// TwinCAT 3 PLC project CM
// ProgramVersion: 3.1.4024.0
// libraries:
//   Tc2_ModbusRTU, * (Beckhoff Automation GmbH)
//   Tc2_Standard, * (Beckhoff Automation GmbH)
//   Tc2_System, * (Beckhoff Automation GmbH)
//   Tc2_Utilities, * (Beckhoff Automation GmbH)
//   Tc3_CM, * (Beckhoff Automation GmbH)
//   Tc3_CM_Base, * (Beckhoff Automation GmbH)
//   Tc3_Filter, * (Beckhoff Automation GmbH)
//   Tc3_Module, * (Beckhoff Automation GmbH)
//   Tc3_MultiArray, * (Beckhoff Automation GmbH)
// project tree:
//   DUTs/ E_AnalysisIDs.TcDUT, ST_HRErrHist.TcDUT
//   FBs/ FB_HRErrHist.TcPOU, FB_SystemTime.TcPOU
//   GVLs/ CM_Params.TcGVL, CM_Data.TcGVL, GVL_ADS.TcGVL, GVL_HMI.TcGVL, GVL_IO.TcGVL
//   / PlcTask.TcTTO, PlcTaskCM.TcTTO, TaskCalc.TcTTO
//   MAIN/ MAIN.TcPOU, MAIN_CM.TcPOU
//   PRGs/ PRG_Calculate.TcPOU, PRG_Database.TcPOU, PRG_Motor_Sensor.TcPOU
// real-time tasks:
//   TASK CMFast: cycle T#1ms, priority 4, ADS port 350
//   TASK CMSlow: cycle T#5ms, priority 12, ADS port 351
//   TASK PMFast: cycle T#1ms, priority 6, ADS port 352
//   TASK PMSlow: cycle T#10ms, priority 16, ADS port 353
//   TASK TaskCalc: cycle T#1ms, priority 8, ADS port 354
//   TASK EIPTask: cycle T#5ms, priority 1, ADS port 301
// I/O:
//   DEVICE Device 5 (EtherCAT) (disabled), AmsNetId 192.168.2.43.6.1
//     Term 1 (EK1100) [EK1100 EtherCAT Coupler (2A E-Bus)]
//       Term 2 (EL1094) [EL1094 4Ch. Dig. Input 24V, 10µs, negative]
//       Term 3 (EL3064) [EL3064 4Ch. Ana. Input 0-10V]
//       Term 4 (EL3632) [EL3632 2Ch. IEPE Sensor]
//       Term 5 (EL6021) [EL6021 Interface (RS422/485)]
//       Term 6 (EL3773) [EL3773 3 Ch. Power Monitoring, Oversample]
//       Term 7 (EL9011) [EL9011 End Terminal]
// variable links:
//   CM/CM Instance <-> Device 5 (EtherCAT)/Term 1 (EK1100)/Term 2 (EL1094)
//     PlcTaskCM Inputs/GVL_IO.bRev <-> Channel 1/Input
//   CM/CM Instance <-> Device 5 (EtherCAT)/Term 1 (EK1100)/Term 3 (EL3064)
//     PlcTaskCM Inputs/GVL_IO.iTemp <-> AI Standard Channel 1/Value
//   CM/CM Instance <-> Device 5 (EtherCAT)/Term 1 (EK1100)/Term 4 (EL3632)
//     PlcTask Inputs/GVL_IO.aEl3632[1][{1..10}] <-> Ch1 Sample {0..9}/Ch1 Value  (10 links)
//   PM/PM Instance <-> Device 5 (EtherCAT)/Term 1 (EK1100)/Term 6 (EL3773)
//     PlcTask Inputs/GVL.stEL3773_1_In/aIL1[10] <-> L1 Current Samples/I1 Samples[9]
//     PlcTask Inputs/GVL.stEL3773_1_In/aIL1[1] <-> L1 Current Samples/I1 Samples[0]
//     PlcTask Inputs/GVL.stEL3773_1_In/aIL1[2] <-> L1 Current Samples/I1 Samples[1]
//     PlcTask Inputs/GVL.stEL3773_1_In/aIL1[3] <-> L1 Current Samples/I1 Samples[2]
//     PlcTask Inputs/GVL.stEL3773_1_In/aIL1[4] <-> L1 Current Samples/I1 Samples[3]
//     PlcTask Inputs/GVL.stEL3773_1_In/aIL1[5] <-> L1 Current Samples/I1 Samples[4]
//     PlcTask Inputs/GVL.stEL3773_1_In/aIL1[6] <-> L1 Current Samples/I1 Samples[5]
//     PlcTask Inputs/GVL.stEL3773_1_In/aIL1[7] <-> L1 Current Samples/I1 Samples[6]
//     PlcTask Inputs/GVL.stEL3773_1_In/aIL1[8] <-> L1 Current Samples/I1 Samples[7]
//     PlcTask Inputs/GVL.stEL3773_1_In/aIL1[9] <-> L1 Current Samples/I1 Samples[8]
//     PlcTask Inputs/GVL.stEL3773_1_In/aIL2[10] <-> L2 Current Samples/I2 Samples[9]
//     PlcTask Inputs/GVL.stEL3773_1_In/aIL2[1] <-> L2 Current Samples/I2 Samples[0]
//     PlcTask Inputs/GVL.stEL3773_1_In/aIL2[2] <-> L2 Current Samples/I2 Samples[1]
//     PlcTask Inputs/GVL.stEL3773_1_In/aIL2[3] <-> L2 Current Samples/I2 Samples[2]
//     PlcTask Inputs/GVL.stEL3773_1_In/aIL2[4] <-> L2 Current Samples/I2 Samples[3]
//     PlcTask Inputs/GVL.stEL3773_1_In/aIL2[5] <-> L2 Current Samples/I2 Samples[4]
//     PlcTask Inputs/GVL.stEL3773_1_In/aIL2[6] <-> L2 Current Samples/I2 Samples[5]
//     PlcTask Inputs/GVL.stEL3773_1_In/aIL2[7] <-> L2 Current Samples/I2 Samples[6]
//     PlcTask Inputs/GVL.stEL3773_1_In/aIL2[8] <-> L2 Current Samples/I2 Samples[7]
//     PlcTask Inputs/GVL.stEL3773_1_In/aIL2[9] <-> L2 Current Samples/I2 Samples[8]
//     PlcTask Inputs/GVL.stEL3773_1_In/aIL3[10] <-> L3 Current Samples/I3 Samples[9]
//     PlcTask Inputs/GVL.stEL3773_1_In/aIL3[1] <-> L3 Current Samples/I3 Samples[0]
//     PlcTask Inputs/GVL.stEL3773_1_In/aIL3[2] <-> L3 Current Samples/I3 Samples[1]
//     PlcTask Inputs/GVL.stEL3773_1_In/aIL3[3] <-> L3 Current Samples/I3 Samples[2]
//     PlcTask Inputs/GVL.stEL3773_1_In/aIL3[4] <-> L3 Current Samples/I3 Samples[3]
//     PlcTask Inputs/GVL.stEL3773_1_In/aIL3[5] <-> L3 Current Samples/I3 Samples[4]
//     PlcTask Inputs/GVL.stEL3773_1_In/aIL3[6] <-> L3 Current Samples/I3 Samples[5]
//     PlcTask Inputs/GVL.stEL3773_1_In/aIL3[7] <-> L3 Current Samples/I3 Samples[6]
//     PlcTask Inputs/GVL.stEL3773_1_In/aIL3[8] <-> L3 Current Samples/I3 Samples[7]
//     PlcTask Inputs/GVL.stEL3773_1_In/aIL3[9] <-> L3 Current Samples/I3 Samples[8]
//     PlcTask Inputs/GVL.stEL3773_1_In/aUL1[10] <-> L1 Voltage Samples/U1 Samples[9]
//     PlcTask Inputs/GVL.stEL3773_1_In/aUL1[1] <-> L1 Voltage Samples/U1 Samples[0]
//     PlcTask Inputs/GVL.stEL3773_1_In/aUL1[2] <-> L1 Voltage Samples/U1 Samples[1]
//     PlcTask Inputs/GVL.stEL3773_1_In/aUL1[3] <-> L1 Voltage Samples/U1 Samples[2]
//     PlcTask Inputs/GVL.stEL3773_1_In/aUL1[4] <-> L1 Voltage Samples/U1 Samples[3]
//     PlcTask Inputs/GVL.stEL3773_1_In/aUL1[5] <-> L1 Voltage Samples/U1 Samples[4]
//     PlcTask Inputs/GVL.stEL3773_1_In/aUL1[6] <-> L1 Voltage Samples/U1 Samples[5]
//     PlcTask Inputs/GVL.stEL3773_1_In/aUL1[7] <-> L1 Voltage Samples/U1 Samples[6]
//     PlcTask Inputs/GVL.stEL3773_1_In/aUL1[8] <-> L1 Voltage Samples/U1 Samples[7]
//     PlcTask Inputs/GVL.stEL3773_1_In/aUL1[9] <-> L1 Voltage Samples/U1 Samples[8]
//     PlcTask Inputs/GVL.stEL3773_1_In/aUL2[10] <-> L2 Voltage Samples/U2 Samples[9]
//     PlcTask Inputs/GVL.stEL3773_1_In/aUL2[1] <-> L2 Voltage Samples/U2 Samples[0]
//     PlcTask Inputs/GVL.stEL3773_1_In/aUL2[2] <-> L2 Voltage Samples/U2 Samples[1]
//     PlcTask Inputs/GVL.stEL3773_1_In/aUL2[3] <-> L2 Voltage Samples/U2 Samples[2]
//     PlcTask Inputs/GVL.stEL3773_1_In/aUL2[4] <-> L2 Voltage Samples/U2 Samples[3]
//     PlcTask Inputs/GVL.stEL3773_1_In/aUL2[5] <-> L2 Voltage Samples/U2 Samples[4]
//     PlcTask Inputs/GVL.stEL3773_1_In/aUL2[6] <-> L2 Voltage Samples/U2 Samples[5]
//     PlcTask Inputs/GVL.stEL3773_1_In/aUL2[7] <-> L2 Voltage Samples/U2 Samples[6]
//     PlcTask Inputs/GVL.stEL3773_1_In/aUL2[8] <-> L2 Voltage Samples/U2 Samples[7]
//     PlcTask Inputs/GVL.stEL3773_1_In/aUL2[9] <-> L2 Voltage Samples/U2 Samples[8]
//     PlcTask Inputs/GVL.stEL3773_1_In/aUL3[10] <-> L3 Voltage Samples/U3 Samples[9]
//     PlcTask Inputs/GVL.stEL3773_1_In/aUL3[1] <-> L3 Voltage Samples/U3 Samples[0]
//     PlcTask Inputs/GVL.stEL3773_1_In/aUL3[2] <-> L3 Voltage Samples/U3 Samples[1]
//     PlcTask Inputs/GVL.stEL3773_1_In/aUL3[3] <-> L3 Voltage Samples/U3 Samples[2]
//     PlcTask Inputs/GVL.stEL3773_1_In/aUL3[4] <-> L3 Voltage Samples/U3 Samples[3]
//     PlcTask Inputs/GVL.stEL3773_1_In/aUL3[5] <-> L3 Voltage Samples/U3 Samples[4]
//     PlcTask Inputs/GVL.stEL3773_1_In/aUL3[6] <-> L3 Voltage Samples/U3 Samples[5]
//     PlcTask Inputs/GVL.stEL3773_1_In/aUL3[7] <-> L3 Voltage Samples/U3 Samples[6]
//     PlcTask Inputs/GVL.stEL3773_1_In/aUL3[8] <-> L3 Voltage Samples/U3 Samples[7]
//     PlcTask Inputs/GVL.stEL3773_1_In/aUL3[9] <-> L3 Voltage Samples/U3 Samples[8]

CONFIGURATION CM
    RESOURCE PLC ON TwinCAT3
        TASK PlcTask(INTERVAL := T#1ms, PRIORITY := 4);
        TASK PlcTaskCM(INTERVAL := T#5ms, PRIORITY := 12);
        TASK TaskCalc(INTERVAL := T#1ms, PRIORITY := 8);
        PROGRAM MAIN WITH PlcTask : MAIN;
        PROGRAM MAIN_CM WITH PlcTaskCM : MAIN_CM;
        PROGRAM PRG_Calculate WITH TaskCalc : PRG_Calculate;
    END_RESOURCE
END_CONFIGURATION

// ---- DUTs/E_AnalysisIDs.TcDUT
TYPE E_AnalysisIDs :
(
	(* analysis chain *)
	eID_Source := 1,
	
	// Magnetude Spectrum
	eID_MagSpectrum,	
	eID_MagSpec_Sink, 
	
	// RMS intergrate
	eID_RMS,	
	eID_RMS_Sink,
	
	// Envelope Spectrum
	eID_EnvSpectrum,	
	eID_EnvSpec_Sink,
	
	// Envelope 
	eID_Env,	
	eID_Env_Sink	
	
) UDINT;
END_TYPE

// ---- DUTs/ST_HRErrHist.TcDUT
TYPE ST_HRErrHist :
STRUCT
{attribute 'displaymode':='hex'}
	hrErrCode	: HRESULT;
	sErrSource	: STRING(63);
	nErrCount	: UDINT;
END_STRUCT
END_TYPE

// ---- GVLs/CM_Params.TcGVL
  VAR_GLOBAL CONSTANT
	cOversamples 		: UDINT 	:= 10;		// number of oversamples
	cMaxChannels		: UDINT		:= 1;
	cOrder				: UDINT		:= 1;		// Maximum order of integration: 0 = acceleration, 1 = velocity, 2 = place. 
	cBufferLength		: UDINT		:= 1600;	// buffer size
	cWindowLength		: UDINT		:= 3200;	// internal buffer size with 50% overlapping
	cRMSBuffer     		: UDINT 	:= 4800;  	// e.g. keep 2 old buffers in mind and add one new buffer to calc RMS value	
	cFFTResult 			: UDINT 	:= 2049;	// result of mag. spectrum (cFFTLength/2+1)
	cFFTLength			: UDINT		:= 4096;	// length of FFT for mag. spectrum	
	cScaleHMI			: UDINT     := 50;
	cWindowParameters	: T_CM_WindowParameters := [0.0, 0.0, 0.0, 0.0, 0.0];	
	
    cInitSource			: ST_MA_MultiArray_InitPars 
						:= ( 	eTypeCode 			:= eMA_TypeCode_LREAL, 
								nDims 				:= 2, 
								aDimSizes 			:= [cMaxChannels,cBufferLength]);	
	
	cInitSpectrum 		: ST_CM_MagnitudeSpectrum_InitPars 
						:= (	nFFT_Length 		:= cFFTLength, 
								nWindowLength 		:= cWindowLength,
								nChannels			:= cMaxChannels,
								bTransformToDecibel	:= FALSE, 
								eWindowType 		:= E_CM_WindowType.eCM_HannWindow, 
								nOverlap			:= cWindowLength/2,
								eScalingType 		:= E_CM_ScalingType.eCM_RMS);
								
	cInitEnvSpec 		: ST_CM_EnvelopeSpectrum_InitPars 
						:= (	nFFT_Length			:= cFFTLength,
								nWindowLength		:= cWindowLength,
								nChannels			:= cMaxChannels,
								bTransformToDecibel	:= FALSE,
								fDecibelThreshold	:= cCM_MinArgLog10, 
								eWindowType			:= eCM_HannWindow,  
								nOverlap			:= cWindowLength/2,         
								eScalingType 		:= eCM_RMS);   
								
	cInitEnv	 		: ST_CM_Envelope_InitPars 
						:= (	nFFT_Length			:= cFFTLength,
								nWindowLength		:= cWindowLength,
								nChannels			:= cMaxChannels);   	
		
	cInitIRMS			: ST_CM_IntegratedRMS_InitPars
						:= ( 	nFFT_Length			:= cFFTLength,
								nWindowLength		:= cWindowLength,
								fSampleRate			:= 10000,
								fLowerFrequencyLimit	:= 20.0,
								fUpperFrequencyLimit	:= 4000.0,
								nMaxBands			:= 1,
								nOrder				:= cOrder,
								nChannels			:= cMaxChannels,
								eWindowType			:= E_CM_WindowType.eCM_HannWindow,
								nOverlap			:=  cWindowLength/2,
								bTransformToDecibel	:= FALSE);
					
END_VAR

VAR_GLOBAL
	fSampleTaskCycleTime		: LREAL := 1; 	// ms
	fSampleRate					: LREAL; 		// Hz  ( sample rate = oversampling factor / cycle time )
	fResolution					: LREAL; 		// Hz/Idx	
	aAccAlarm					: ARRAY[1..cMaxChannels] OF LREAL;
	aVeloAlarm					: ARRAY[1..cMaxChannels] OF LREAL;
	aEnvAlarm					: ARRAY[1..cMaxChannels] OF LREAL;
	
	aAccWarning					: ARRAY[1..cMaxChannels] OF LREAL;
	aVeloWarning				: ARRAY[1..cMaxChannels] OF LREAL;
	aEnvWarning					: ARRAY[1..cMaxChannels] OF LREAL;
	
	nCurrentDate				: WORD;
	sCurrentTime				: STRING;
	nCurrentHour				: WORD;
	nCurrentSec					: WORD;
	
END_VAR

// ---- GVLs/CM_Data.TcGVL
VAR_GLOBAL

	aAccBuffer			: ARRAY[1..cMaxChannels] OF ARRAY[1..cOversamples] OF LREAL;   	
		
	aMagSpecResult		: ARRAY[1..cMaxChannels] OF ARRAY[1..cFFTResult] OF LREAL;	
	aVeloSpecResult		: ARRAY[1..cMaxChannels] OF ARRAY[1..cFFTResult] OF LREAL;
	aEnvSpecResult		: ARRAY[1..cMaxChannels] OF ARRAY[1..cFFTResult] OF LREAL;
	
	aEnvResult			: ARRAY[1..cMaxChannels] OF ARRAY[1..cBufferLength] OF LREAL;
		
	aRMSResult			: ARRAY[1..cMaxChannels] OF ARRAY[1..cOrder+1] OF LREAL;
	aRMSEnvResult		: ARRAY[1..cMaxChannels] OF LREAL;

	fFrequency			: ARRAY[1..cMaxChannels] OF ARRAY[1..cFFTResult] OF LREAL; 		// Hz	
	aTWFBuffer			: ARRAY[1..cMaxChannels] OF ARRAY[1..cOversamples*cScaleHMI] OF LREAL;  
	aTime				: ARRAY[1..cOversamples*cScaleHMI] OF UDINT;	
END_VAR

// ---- GVLs/GVL_ADS.TcGVL
VAR_GLOBAL
	aFFTAcceleration1Add 	: ARRAY[1..cFFTResult] OF LREAL;
	aFFTVelocity1Add 		: ARRAY[1..cFFTResult] OF LREAL;
	aFFTEnvelope1Add 		: ARRAY[1..cFFTResult] OF LREAL;
	RMSAcc1Add				: LREAL;
	RMSVel1Add				: LREAL;
	RMSEnv1Add				: LREAL;
	Temperature1Add			: REAL;
	//point_2
	aFFTAcceleration2Add 	: ARRAY[1..cFFTResult] OF LREAL;
	aFFTVelocity2Add 		: ARRAY[1..cFFTResult] OF LREAL;
	aFFTEnvelope2Add 		: ARRAY[1..cFFTResult] OF LREAL;
	RMSAcc2Add				: LREAL;
	RMSVel2Add				: LREAL;
	RMSEnv2Add				: LREAL;
	Temperature2Add			: REAL;
	//bAdd
	bAddData				: BOOL;
	bCheckADS				: BOOL;
	bError					: BOOL;
END_VAR

// ---- GVLs/GVL_HMI.TcGVL
VAR_GLOBAL
	//Read
	Output_frequency_monitor			: REAL;//Hz
	UpperLimit_frequency_monitor		: REAL; //Hz
	Power_on_time_monitor				: INT;	//Hour	
	Output_current_monitor				: REAL;//A
	Rotation_direction_monitor			: STRING;//o: Stop d: 0Hz output F: Forward r: Reverse
	Inverter_Temperature				: REAL;//C 
	Inverter_Voltage_Output				: REAL;//V
	//Write
	Run_Motor							: BOOL;
	Rotation_direction					: BOOL;
	Frequence							: REAL;//Hz
	Acceleration_time					: REAL;//s
	Deceleration_time					: REAL;//s
	//read terminal
	iActSpeed							: INT;
	Temperature_motor					: REAL;
END_VAR

// ---- GVLs/GVL_IO.TcGVL
VAR_GLOBAL
	aEl3632 AT %I*		: ARRAY[1..cMaxChannels] OF ARRAY[1..cOversamples] OF INT;	// Input from hardware e.g. EL3632	
	wMotorRun	AT %Q*	: WORD;
	wFreq		AT %Q*	: WORD;
	bRev		AT %I*	: BOOL;
	iTemp		AT %I*	: INT;
	bMotorRun			: BOOL;
	fFreq				: REAL;
END_VAR

// ---- MAIN/MAIN.TcPOU
PROGRAM MAIN
VAR
	nSample				: UDINT;
	
	fbSource			: FB_CMA_Source := (	stInitPars 	:= cInitSource, 
												nOwnID 		:= eID_Source, 
												aDestIDs 	:= [eID_MagSpectrum,
																eID_EnvSpectrum,
																eID_Env,
																eID_RMS]);		
										
	fbSinkMagSpec		: FB_CMA_Sink 	:= ( 	nOwnID 		:= eID_MagSpec_Sink);
	fbSinkEnvSpec		: FB_CMA_Sink 	:= ( 	nOwnID 		:= eID_EnvSpec_Sink);
	fbSinkEnv			: FB_CMA_Sink 	:= ( 	nOwnID 		:= eID_Env_Sink);
	fbSinkRMS			: FB_CMA_Sink 	:= ( 	nOwnID 		:= eID_RMS_Sink); 
	
	nChannelIdx			: UDINT;

	k, m, l: UDINT;
	nChnIdx: UDINT;
END_VAR

Source();
Sink();
// input from EL3632
FOR nChannelIdx := 1 TO cMaxChannels DO
	FOR k := 1 TO cOversamples DO
		aAccBuffer[nChannelIdx][k] 		:= INT_TO_LREAL(aEl3632[nChannelIdx][k])*(5/EXPT(2,15))/(0.1)*9.81;
	END_FOR	
END_FOR

ACTION Sink:
// Push results to sink

fbSinkMagSpec.Output2DStd(	pDataOut 	:= ADR(aMagSpecResult), 
					nDataOutSize 		:= SIZEOF(aMagSpecResult), 
					eElementType 		:= eMA_TypeCode_LREAL, 
					nOptionPars			:= 0);
				
fbSinkEnvSpec.Output2DStd(	pDataOut 	:= ADR(aEnvSpecResult), 
					nDataOutSize 		:= SIZEOF(aEnvSpecResult), 
					eElementType 		:= eMA_TypeCode_LREAL, 
					nOptionPars			:= 0); 
					
fbSinkEnv.Output2DStd(	pDataOut 		:= ADR(aEnvResult), 
					nDataOutSize 		:= SIZEOF(aEnvResult), 
					eElementType 		:= eMA_TypeCode_LREAL, 
					nOptionPars			:= 0); 								
				
fbSinkRMS.Output2DStd(	pDataOut 		:= ADR(aRMSResult), 
					nDataOutSize 		:= SIZEOF(aRMSResult), 
					eElementType 		:= eMA_TypeCode_LREAL, 
					nOptionPars			:= 0);
END_ACTION

ACTION Source:
fbSource.Input2DStd( pDataIn 			:= ADR(aAccBuffer),
				  nDataInSize 			:= SIZEOF(aAccBuffer), 
				  eElementType 			:= eMA_TypeCode_LREAL,
				  nOptionPars			:= cCMA_Option_MarkInterruption );
END_ACTION

END_PROGRAM

// ---- MAIN/MAIN_CM.TcPOU
PROGRAM MAIN_CM
VAR
	fbMagSpec			: FB_CMA_MagnitudeSpectrum 
						:= (	stInitPars 	:= cInitSpectrum, 
								nOwnID 		:= eID_MagSpectrum, 
								aDestIDs 	:= [eID_MagSpec_Sink] ); 
										
	fbEnvSpec			: FB_CMA_EnvelopeSpectrum 
						:= ( 	stInitPars 	:= cInitEnvSpec, 
								nOwnID 		:= eID_EnvSpectrum, 
								aDestIDs 	:= [eID_EnvSpec_Sink] );	
								
	fbEnv				: FB_CMA_Envelope 
						:= ( 	stInitPars 	:= cInitEnv, 
								nOwnID 		:= eID_Env, 
								aDestIDs 	:= [eID_Env_Sink] );	
								
	fbRMS				: FB_CMA_IntegratedRMS
						:= ( 	stInitPars	:= cInitIRMS,
								nOwnID		:= eID_RMS,
								aDestIDs	:= [eID_RMS_Sink]);
		
	nErrorID			: UDINT;
	fbErrHist			: FB_HRErrHist; 
	hrErrList			: ARRAY[1..2] OF HRESULT;
	bPause				: BOOL;
	
END_VAR

IF NOT bPause THEN
//
END_IF

PRG_Database();
PRG_Motor_Sensor();

fbMagSpec.Call();
fbEnvSpec.Call();
fbEnv.Call();

fbRMS.Call();
//fbHistArray.CallEx(nAppendData := cAppendData, bResetData := bResetHist);

END_PROGRAM

// ---- FBs/FB_HRErrHist.TcPOU
FUNCTION_BLOCK FB_HRErrHist
(* v1.10
build up an error history consisting of two arrays and one index.
The index shows the actual array position. The last error id and the count for this id are saved in the arrays.
If an error id is the same as the previous input error the counter is increased. Otherwise the index is increased.
*)
VAR_INPUT
	bEdgeDetect	: BOOL;	(* FALSE: every input(bErr) is processed; TRUE: only rising edge of input is processed *)
END_VAR
VAR_OUTPUT
	nErrSum		: UINT;
	nErrIdx		: UINT; // error list index of last occured error (max. cHistLen)
	aErrList	: ARRAY[1..cHistLen] OF ST_HRErrHist;
END_VAR

VAR
	bNewErr		: BOOL;
	fbErrTrig	: R_TRIG;
END_VAR
VAR CONSTANT
	cHistLen	: UINT := 100;
END_VAR

METHOD AddError
VAR_INPUT
	bErr		: BOOL;
	hrErrCode	: HRESULT;
	sErrSource	: STRING(63);
END_VAR
fbErrTrig(CLK:=bErr);
IF bEdgeDetect THEN
	bNewErr := fbErrTrig.Q;
ELSE
	bNewErr := bErr;
END_IF

IF bNewErr THEN
	nErrSum := nErrSum + 1;
	IF nErrIdx < cHistLen THEN
		IF nErrIdx = 0 THEN
			nErrIdx	:= nErrIdx + 1;
		ELSIF aErrList[nErrIdx].hrErrCode <> hrErrCode OR aErrList[nErrIdx].sErrSource <> sErrSource THEN
			nErrIdx	:= nErrIdx + 1;
		END_IF
		aErrList[nErrIdx].hrErrCode := hrErrCode;
		aErrList[nErrIdx].sErrSource := sErrSource;
		aErrList[nErrIdx].nErrCount := aErrList[nErrIdx].nErrCount + 1;
	END_IF
END_IF
END_METHOD

METHOD Reset
VAR_INPUT
END_VAR
nErrSum := 0;
nErrIdx := 0;
MEMSET(ADR(aErrList),0,SIZEOF(aErrList));
END_METHOD

END_FUNCTION_BLOCK

// ---- PRGs/PRG_Database.TcPOU
PROGRAM PRG_Database
VAR
	fbSystemTime			:	FB_SystemTime;
	bSaveData				: BOOL;
	bLoadData				: BOOL;
	nStateSave, nStateLoad	: INT;
	tTimer1, tTimer2		: TON;
	bTest					: BOOL;
	nStateADS				: INT;
END_VAR

fbSystemTime();
sCurrentTime	:= fbSystemTime.sTime;
nCurrentSec		:= fbSystemTime.wSecond;
CASE nStateSave OF
	0:
		tTimer1(IN := FALSE);
		IF nCurrentSec = 70 OR sCurrentTime = '06:00:00' OR sCurrentTime = '14:00:00' OR sCurrentTime = '22:00:00' THEN
			nStateSave			:= 1;
		END_IF
	1:
		aFFTAcceleration1Add		:= aMagSpecResult[1];
		aFFTVelocity1Add			:= aVeloSpecResult[1];
		aFFTEnvelope1Add			:= aEnvSpecResult[1];
		RMSAcc1Add					:= aRMSResult[1][1]/9.81;
		RMSVel1Add					:= aRMSResult[1][2]*1000;
		RMSEnv1Add					:= aRMSEnvResult[1]/9.81;
(*		
		aFFTAcceleration2Add		:= aMagSpecResult[2];
		aFFTVelocity2Add			:= aVeloSpecResult[2];
		aFFTEnvelope2Add			:= aEnvSpecResult[2];
		RMSAcc2Add					:= aRMSResult[2][1]/9.81;
		RMSVel2Add					:= aRMSResult[2][2]*1000;
		RMSEnv2Add					:= aRMSEnvResult[2]/9.81;		*)
		bAddData					:= TRUE;
		nStateSave					:= 2;
	2:
		IF NOT bAddData THEN
			tTimer1(IN := TRUE,PT := T#2S);
			IF tTimer1.Q THEN
				nStateSave			:= 0;		
			END_IF	
		END_IF
			
		
END_CASE

CASE nStateADS OF
	0:
		IF bCheckADS THEN
			nStateADS := 1;
		ELSE
			tTimer2(IN := TRUE,PT := T#5S);
			IF tTimer2.Q THEN
				nStateADS := 2;
			END_IF
		END_IF
		
	1:
		bCheckADS := FALSE;
		bError	:= FALSE;
		tTimer2(IN := FALSE);
		nStateADS := 0;
	2:
		bError := TRUE;
		tTimer2(IN := FALSE);
		IF bCheckADS THEN
			nStateADS := 0;
		END_IF
END_CASE

END_PROGRAM

// ---- FBs/FB_SystemTime.TcPOU
FUNCTION_BLOCK FB_SystemTime
VAR_INPUT
END_VAR
VAR_OUTPUT
END_VAR
VAR
	GetLocalSystemTime 	: FB_LocalSystemTime;
	wDateW				: WORD;
END_VAR

GetLocalSystemTime(bEnable := TRUE);

PROPERTY dtDateTimeFull : DT
GET
dtDateTimeFull 	:= SYSTEMTIME_TO_DT(GetLocalSystemTime.systemTime);
END_GET
END_PROPERTY

PROPERTY sDate : STRING
GET
sDate	:= MID(sDateTimeFull,10,1);
END_GET
END_PROPERTY

PROPERTY sDateTime : STRING
GET
sDateTime := MID(sDateTimeFull,19,1);
END_GET
END_PROPERTY

PROPERTY sDateTimeFull : STRING
GET
sDateTimeFull 	:= SYSTEMTIME_TO_STRING(GetLocalSystemTime.systemTime);
END_GET
END_PROPERTY

PROPERTY sDayOfWeek : STRING
GET
wDateW	:=  GetLocalSystemTime.systemTime.wDayOfWeek;
IF wDateW = 0 THEN
	sDayOfWeek := 'Sunday';
ELSIF wDateW = 1 THEN
	sDayOfWeek := 'Monday';
ELSIF wDateW = 2 THEN
	sDayOfWeek := 'Tuesday';
ELSIF wDateW = 3 THEN
	sDayOfWeek := 'Wednesday';
ELSIF wDateW = 4 THEN
	sDayOfWeek := 'Thursday';
ELSIF wDateW = 5 THEN
	sDayOfWeek := 'Friday';
ELSIF wDateW = 6 THEN
	sDayOfWeek := 'Saturday';
END_IF
END_GET
END_PROPERTY

PROPERTY sTime : STRING
GET
sTime := MID(sDateTimeFull,8,12);
END_GET
END_PROPERTY

PROPERTY wDay : Word
GET
wDay :=  GetLocalSystemTime.systemTime.wDay;
END_GET
END_PROPERTY

PROPERTY wHour : WORD
GET
wHour	:=	GetLocalSystemTime.systemTime.wHour;
END_GET
END_PROPERTY

PROPERTY wMilliSeconds : WORD
GET
wMilliseconds	:=	GetLocalSystemTime.systemTime.wMilliseconds;
END_GET
END_PROPERTY

PROPERTY wMinute : WORD
GET
wMinute	:=	GetLocalSystemTime.systemTime.wMinute;
END_GET
END_PROPERTY

PROPERTY wMonth : Word
GET
wMonth	:=  GetLocalSystemTime.systemTime.wMonth;
END_GET
END_PROPERTY

PROPERTY wSecond : WORD
GET
wSecond	:=	GetLocalSystemTime.systemTime.wSecond;
END_GET
END_PROPERTY

PROPERTY wYear : Word
GET
wYear :=  GetLocalSystemTime.systemTime.wYear;
END_GET
END_PROPERTY

END_FUNCTION_BLOCK

// ---- PRGs/PRG_Motor_Sensor.TcPOU
PROGRAM PRG_Motor_Sensor
VAR
	//Motor read
	state_mt	: INT;
	Data_mt_1	: ARRAY[0..2] OF INT;//0:Output_frequency_monitor 1:Output_current_monitor 2:Rotation_direction_monitor
	Data_mt_2	: INT;//temperature
	Data_mt_3	: INT;//voltage
	Data_mt_4	: INT;//Power_on - hour 
	Data_mt_5	: INT;//Limit Frequency
	//Motor write
	run_temp 							: BOOL;
	Rotation_direction_temp				: BOOL;
	Frequence_temp						: REAL;//Hz
	Acceleration_time_temp				: REAL;//s
	Deceleration_time_temp				: REAL;//s
	//Datawrite_mt_1						: ARRAY[0..1] OF BOOL;
	Datawrite_mt_2						: INT;//Frequence
	Datawrite_mt_3						: ARRAY[0..3] OF INT;//acc vs dec
	// Sensor
	Rev_T		: R_TRIG;
	state_ss	: INT;
	pulse		: INT;
	i			: INT := 1;
	data		: INT;
	rpm			: REAL;
	timer		: TON;
	fb_Modbus	: ModbusRtuMaster_KL6x22B;
END_VAR

Motor();
Sensor();
Output_frequency_monitor			:= INT_TO_REAL(Data_mt_1[0])/100;//Hz
Output_current_monitor				:= INT_TO_REAL(Data_mt_1[1])/100;//A
IF (Data_mt_1[2] = 0) THEN
	Rotation_direction_monitor		:= 'Stop';
ELSIF (Data_mt_1[2] = 1) THEN			
	Rotation_direction_monitor		:= '0Hz';
ELSIF (Data_mt_1[2] = 2) THEN
	Rotation_direction_monitor		:= 'Forward';
ELSIF (Data_mt_1[2] = 3) THEN
	Rotation_direction_monitor		:= 'Reverse';
END_IF
Inverter_Temperature				:= INT_TO_REAL(Data_mt_2)/10;//C
Inverter_Voltage_Output				:= INT_TO_REAL(Data_mt_3)/10;//V
Power_on_time_monitor				:= Data_mt_4;//hour
UpperLimit_frequency_monitor		:= INT_TO_REAL(Data_mt_5)/100;//V

ACTION Motor:
CASE state_mt OF
	0://init
			run_temp					:= Run_Motor;
			Rotation_direction_temp		:= Rotation_direction;
			Frequence_temp				:= Frequence;
			Acceleration_time_temp		:= Acceleration_time;
			Deceleration_time_temp		:= Deceleration_time;
			state_mt 					:= 1;
	1://read data1
		fb_Modbus.ReadRegs(
				UnitID:= 1, 
				Quantity:= 3, 
				MBAddr:= 10000, 
				cbLength:= SIZEOF(Data_mt_1), 
				pMemoryAddr:= ADR(Data_mt_1), 
				Execute:= TRUE, 
				Timeout:= T#1S, 
				BUSY=> , 
				Error=> , 
				ErrorId=> , 
				cbRead=> ); 
		IF NOT fb_Modbus.BUSY AND NOT fb_Modbus.Error THEN
			fb_Modbus.ReadRegs(Execute:= FALSE); 
			state_mt 			:= 2;
		END_IF
	2://read data2
		fb_Modbus.ReadRegs(
			UnitID:= 1, 
			Quantity:= 1, 
			MBAddr:= 10214, 
			cbLength:= SIZEOF(Data_mt_2), 
			pMemoryAddr:= ADR(Data_mt_2), 
			Execute:= TRUE, 
			Timeout:= T#1S, 
			BUSY=> , 
			Error=> , 
			ErrorId=> , 
			cbRead=> );
		IF NOT fb_Modbus.BUSY AND NOT fb_Modbus.Error THEN
			fb_Modbus.ReadRegs(Execute:= FALSE);
			state_mt 			:= 3;
		END_IF
	3://read data3
		fb_Modbus.ReadRegs(
			UnitID:= 1, 
			Quantity:= 1, 
			MBAddr:= 10017, 
			cbLength:= SIZEOF(Data_mt_3), 
			pMemoryAddr:= ADR(Data_mt_3), 
			Execute:= TRUE, 
			Timeout:= T#1S, 
			BUSY=> , 
			Error=> , 
			ErrorId=> , 
			cbRead=> );
		IF NOT fb_Modbus.BUSY AND NOT fb_Modbus.Error THEN
			fb_Modbus.ReadRegs(Execute:= FALSE);
			state_mt 			:= 4;
		END_IF
	4://read data4
		fb_Modbus.ReadRegs(
			UnitID:= 1, 
			Quantity:= 1, 
			MBAddr:= 10224, 
			cbLength:= SIZEOF(Data_mt_4), 
			pMemoryAddr:= ADR(Data_mt_4), 
			Execute:= TRUE, 
			Timeout:= T#1S, 
			BUSY=> , 
			Error=> , 
			ErrorId=> , 
			cbRead=> );
		IF NOT fb_Modbus.BUSY AND NOT fb_Modbus.Error THEN
			fb_Modbus.ReadRegs(Execute:= FALSE);
			state_mt 			:= 5;
		END_IF
	5://read data4
		fb_Modbus.ReadRegs(
			UnitID:= 1, 
			Quantity:= 1, 
			MBAddr:= 10013, 
			cbLength:= SIZEOF(Data_mt_5), 
			pMemoryAddr:= ADR(Data_mt_5), 
			Execute:= TRUE, 
			Timeout:= T#1S, 
			BUSY=> , 
			Error=> , 
			ErrorId=> , 
			cbRead=> );
		IF NOT fb_Modbus.BUSY AND NOT fb_Modbus.Error THEN
			fb_Modbus.ReadRegs(Execute:= FALSE);
			state_mt 			:= 6;
		END_IF
	6://check write run
		IF (Run_Motor <> run_temp) THEN
			state_mt 			:= 60;//write run
		ELSE
			state_mt 			:= 7;
		END_IF
	7:// check frequence
		IF (Frequence <> Frequence_temp) THEN
			state_mt 			:= 70;//write frequence
		ELSE
			state_mt 			:= 8;
		END_IF
	8://check Acc vs Dec time
		IF (Acceleration_time <> Acceleration_time_temp) OR (Deceleration_time <> Deceleration_time_temp) THEN
			state_mt 			:= 80;//write acc and dec
		ELSE
			state_mt 			:= 9; 
		END_IF
	9://
		IF (Rotation_direction <> Rotation_direction_temp) THEN
			state_mt 			:= 90;
		ELSE
			state_mt 			:= 1;
		END_IF
	//=============================================
	60://write run
		fb_Modbus.WriteSingleCoil(
			UnitID:= 1, 
			Quantity:= 1, 
			MBAddr:= 0, 
			cbLength:= SIZEOF(Run_Motor), 
			pMemoryAddr:= ADR(Run_Motor), 
			Execute:= TRUE, 
			Timeout:= T#1S, 
			BUSY=> , 
			Error=> , 
			ErrorId=> , 
			cbRead=> );
		IF NOT fb_Modbus.BUSY AND NOT fb_Modbus.Error THEN
			fb_Modbus.WriteSingleCoil(Execute := FALSE);
			run_temp							 := Run_Motor;
			state_mt 							 := 7;//return
		END_IF
	70://write Freq
		Datawrite_mt_2 := REAL_TO_INT(Frequence*100);
		fb_Modbus.WriteRegs(
			UnitID:= 1, 
			Quantity:= 1, 
			MBAddr:= 11000, 
			cbLength:= SIZEOF(Datawrite_mt_2), 
			pMemoryAddr:= ADR(Datawrite_mt_2), 
			Execute:= TRUE, 
			Timeout:= T#1S, 
			BUSY=> , 
			Error=> , 
			ErrorId=> , 
			cbRead=> );
		IF NOT fb_Modbus.BUSY AND NOT fb_Modbus.Error THEN
			fb_Modbus.WriteRegs(Execute := FALSE);
			Frequence_temp				:= Frequence;
			state_mt 					:= 8;//return
		END_IF
	80://write acc vs dec
		Datawrite_mt_3[0] := REAL_TO_INT(Acceleration_time*100);
		Datawrite_mt_3[1] := 0;
		Datawrite_mt_3[2] := REAL_TO_INT(Deceleration_time_temp*100);
		Datawrite_mt_3[3] := 0;
		fb_Modbus.WriteRegs(
			UnitID:= 1, 
			Quantity:= 4, 
			MBAddr:= 11010, 
			cbLength:= SIZEOF(Datawrite_mt_3), 
			pMemoryAddr:= ADR(Datawrite_mt_3), 
			Execute:= TRUE, 
			Timeout:= T#1S, 
			BUSY=> , 
			Error=> , 
			ErrorId=> , 
			cbRead=> );
		IF NOT fb_Modbus.BUSY AND NOT fb_Modbus.Error THEN
			fb_Modbus.WriteRegs(Execute := FALSE);
			Acceleration_time_temp		:= Acceleration_time;
			Deceleration_time_temp		:= Deceleration_time;
			state_mt 					:= 9;
		END_IF
	90://
		fb_Modbus.WriteSingleCoil(
			UnitID:= 1, 
			Quantity:= 1, 
			MBAddr:= 1, 
			cbLength:= SIZEOF(Rotation_direction), 
			pMemoryAddr:= ADR(Rotation_direction), 
			Execute:= TRUE, 
			Timeout:= T#1S, 
			BUSY=> , 
			Error=> , 
			ErrorId=> , 
			cbRead=> );
		IF NOT fb_Modbus.BUSY AND NOT fb_Modbus.Error THEN
			fb_Modbus.WriteSingleCoil(Execute := FALSE);
			Rotation_direction_temp				 := Rotation_direction;
			state_mt 							 := 1;//return
		END_IF
END_CASE
END_ACTION

ACTION Sensor:
Rev_T( CLK := bRev);
IF Rev_T.Q THEN
	pulse	:= pulse + 1;	
END_IF
CASE state_ss OF
	0:
		timer( IN := TRUE, PT := T#1S);
		IF timer.Q THEN
			data  := pulse;
			timer( IN := FALSE);
			state_ss := 1;
		END_IF
	1:
		rpm	:= data*60;
		pulse	:= 0;
		state_ss := 0;
END_CASE
iActSpeed	:= REAL_TO_INT(rpm);
END_ACTION

END_PROGRAM

// ---- PRGs/PRG_Calculate.TcPOU
PROGRAM PRG_Calculate
VAR
	nChnIdx, i, k		: UDINT;
	m, n, p, j, l, q	: UDINT:= 1;
	fSumRMSEnv			: LREAL;
END_VAR

FOR nChnIdx := 1 TO cMaxChannels DO
	// Calculate Frequency
	fSampleRate								:= cOversamples * (1000.0 / fSampleTaskCycleTime);
	fResolution 							:= fSampleRate / cFFTLength;	
	
	// Calculate velocity spectrum                              	     	
	FOR i := 1 TO cFFTResult DO             	
		fFrequency[nChnIdx][i]				:= (i - 1) * fResolution;			
		IF i <> 1 THEN
			aVeloSpecResult[nChnIdx][i]		:= aMagSpecResult[nChnIdx][i]/(2*PI*fFrequency[nChnIdx][i])*1000;
		ELSE
			aVeloSpecResult[nChnIdx][i]		:= 0;
		END_IF
	END_FOR
	
	//Calculate RMS of Envelope
	fSumRMSEnv 								:= 0;
	FOR p := 1 TO cBufferLength DO
		fSumRMSEnv							:= fSumRMSEnv + EXPT(aEnvResult[nChnIdx][p],2);
	END_FOR
	aRmsEnvResult[nChnIdx]					:= SQRT(fSumRMSEnv/cBufferLength);
	
	//Scale up for HMI 
	IF m < cScaleHMI THEN
		FOR n := 1 TO cOversamples DO
			aTWFBuffer[nChnIdx][(m-1)*10+n]		:= aAccBuffer[nChnIdx][n];   
		END_FOR
		m										:= m + 1;
	ELSE
		m										:= cScaleHMI;
		FOR l := 1 TO cScaleHMI-1 DO
			FOR n := 1 TO cOversamples DO
				aTWFBuffer[nChnIdx][(l-1)*10+n]	:= aTWFBuffer[nChnIdx][(l)*10+n];   
			END_FOR
		END_FOR
		FOR q := 1 TO cOversamples DO
			aTWFBuffer[nChnIdx][(m-1)*10+q]		:= aAccBuffer[nChnIdx][q];   
		END_FOR	
	END_IF	
	
END_FOR

IF aTime[cOversamples*cScaleHMI] <> cOversamples*cScaleHMI THEN
	FOR k := 1 TO cOversamples*cScaleHMI DO aTime[k] := k; END_FOR
END_IF

END_PROGRAM
